// TIA Portal V21 export
TYPE "UDT_Settings"
   STRUCT
      AlarmDelays : Struct
         Protection : Time;
         Communication : Time;
         DriveFault : Time;
         LowCurrent : Time;
         WorkConfirmation : Time;
         Tank : Time := T#5m;
         Sensor { ExternalAccessible := 'False'; ExternalVisible := 'False'; ExternalWritable := 'False'} : Time;
      END_STRUCT;
      Sensors : Struct
         LiquidLevel : Struct
            Tank_1 : "AnalogInputSettings";
            Tank_2 : "AnalogInputSettings";
         END_STRUCT;
      END_STRUCT;
   END_STRUCT;
END_TYPE
